IF (VI_Severity <> L_Last_Severity) OR (VI_RootCause <> L_Last_RootCause) THEN
    CASE VI_RootCause OF
        E_System_Root_Cause.ROOT_FIRE:
            L_Event_Text := 'EVENT: FIRE DETECTED';
        E_System_Root_Cause.ROOT_GAS_LEAK:
            L_Event_Text := 'EVENT: GAS LEAK';
        E_System_Root_Cause.ROOT_CO_CRITICAL:
            L_Event_Text := 'EVENT: CO CRITICAL';
        E_System_Root_Cause.ROOT_CO_WARNING:
            L_Event_Text := 'EVENT: CO WARNING';
        E_System_Root_Cause.ROOT_WATER_LEAK:
            L_Event_Text := 'EVENT: WATER LEAK';
        E_System_Root_Cause.ROOT_SENSOR_FAULT:
            L_Event_Text := 'EVENT: SENSOR FAULT';
        E_System_Root_Cause.ROOT_IO_OFFLINE:
            L_Event_Text := 'EVENT: IO OFFLINE';
        E_System_Root_Cause.ROOT_COMM_FAULT:
            L_Event_Text := 'EVENT: COMM FAULT';
        E_System_Root_Cause.ROOT_WATCHDOG_FAULT:
            L_Event_Text := 'EVENT: WATCHDOG FAULT';
        E_System_Root_Cause.ROOT_SUBSYSTEM_FAULT:
            L_Event_Text := 'EVENT: SUBSYSTEM FAULT';
        ELSE
            L_Event_Text := 'EVENT: SYSTEM STATE CHANGE';
    END_CASE;

    L_Write_Index := L_Write_Index + 1;
    IF L_Write_Index > 16 THEN
        L_Write_Index := 1;
    END_IF;

    VO_Event_Time_MS[L_Write_Index] := VI_Time_MS;
    VO_Event_Severity[L_Write_Index] := VI_Severity;
    VO_Event_RootCause[L_Write_Index] := VI_RootCause;
    VO_Event_Text[L_Write_Index] := L_Event_Text;

    VO_Last_Index := L_Write_Index;
    VO_Last_Event_Text := L_Event_Text;

    IF VO_Event_Count < 16 THEN
        VO_Event_Count := VO_Event_Count + 1;
    END_IF;
END_IF;

L_Last_Severity := VI_Severity;
L_Last_RootCause := VI_RootCause;
// >>> BULK_SYNC_ANCHOR: FB_Fault_Logger <<<

          
END_FUNCTION_BLOCK

FUNCTION_BLOCK FB_HMI_Interface
  VAR_INPUT
    VI_System_Time_MS : UDINT;
    VI_Latitude : REAL := 55.75;  (* Москва *)
    VI_Longitude : REAL := 37.61;
  END_VAR
  VAR_OUTPUT
    VO_Sunset_Time : TOD;
    VO_Sunrise_Time : TOD;
    VO_Is_Night : BOOL;
  END_VAR
  VAR
    L_Current_TOD : TOD;
  END_VAR

            FUNCTION_BLOCK FB_HMI_Interface
VAR_INPUT
    VI_Severity   : E_System_Severity;
    VI_RootCause  : E_System_Root_Cause;
    VI_Status_Msg : STRING(200);
END_VAR

VAR_OUTPUT
    VO_HMI_Status_Text : STRING(200);
    VO_HMI_State_Code  : INT;
END_VAR

VO_HMI_Status_Text := VI_Status_Msg;

CASE VI_Severity OF
    E_System_Severity.SEV_NORMAL:
        VO_HMI_State_Code := 0;
    E_System_Severity.SEV_WARNING:
        VO_HMI_State_Code := 1;
    E_System_Severity.SEV_DEGRADED:
        VO_HMI_State_Code := 2;
    E_System_Severity.SEV_CRITICAL:
        VO_HMI_State_Code := 3;
END_CASE;
// >>> BULK_SYNC_ANCHOR: FB_HMI_Interface <<<

          
END_FUNCTION_BLOCK

FUNCTION_BLOCK FB_IO_Module_Watchdog
  VAR_INPUT
    VI_System_Time_MS : UDINT;
    VI_Latitude : REAL := 55.75;  (* Москва *)
    VI_Longitude : REAL := 37.61;
  END_VAR
  VAR_OUTPUT
    VO_Sunset_Time : TOD;
    VO_Sunrise_Time : TOD;
    VO_Is_Night : BOOL;
  END_VAR
  VAR
    L_Current_TOD : TOD;
  END_VAR

            FUNCTION_BLOCK FB_IO_Module_Watchdog
VAR_INPUT
    VI_System_Time_MS : UDINT;
    VI_Module_ID : BYTE;
    VI_Heartbeat_Signal : BOOL; // Сигнал от модуля (например, мигающий бит)
    VI_Timeout_MS : UDINT := 2000; // Таймаут 2 секунды по умолчанию
END_VAR
VAR_OUTPUT
    VO_Module_Online : BOOL;
    VO_Error_Active : BOOL;
END_VAR
VAR
    L_Last_Heartbeat_State : BOOL;
    L_Last_Heartbeat_Time : UDINT;
    L_Elapsed_Time : UDINT;
END_VAR

// Отслеживание изменения сигнала
IF VI_Heartbeat_Signal <> L_Last_Heartbeat_State THEN
    L_Last_Heartbeat_Time := VI_System_Time_MS;
    L_Last_Heartbeat_State := VI_Heartbeat_Signal;
END_IF;

// Проверка таймаута
L_Elapsed_Time := F_TimeDiff(VI_System_Time_MS, L_Last_Heartbeat_Time);

IF L_Elapsed_Time > VI_Timeout_MS THEN
    VO_Module_Online := FALSE;
    VO_Error_Active := TRUE;
ELSE
    VO_Module_Online := TRUE;
    VO_Error_Active := FALSE;
END_IF;
// >>> BULK_SYNC_ANCHOR: FB_IO_Module_Watchdog <<<

          
END_FUNCTION_BLOCK

FUNCTION_BLOCK FB_Redundancy_Manager
  VAR_INPUT
    VI_System_Time_MS : UDINT;
    VI_Latitude : REAL := 55.75;  (* Москва *)
    VI_Longitude : REAL := 37.61;
  END_VAR
  VAR_OUTPUT
    VO_Sunset_Time : TOD;
    VO_Sunrise_Time : TOD;
    VO_Is_Night : BOOL;
  END_VAR
  VAR
    L_Current_TOD : TOD;
  END_VAR

            FUNCTION_BLOCK FB_Redundancy_Manager
VAR_INPUT
    VI_System_Time_MS : UDINT; // Системное время (мс)
    VI_Local_PLC_ID : BYTE; // 1 = ПЛК А, 2 = ПЛК B
    VI_Remote_Pulse : BOOL; // Сигнал от партнера
    VI_Remote_Is_Active : BOOL; // Статус партнера
    VI_Gateway_Ping_OK : BOOL; // Пинг до шлюза
    VI_Remote_State : ST_System_State_Snapshot; // Состояние партнера
    VI_Local_State : ST_System_State_Snapshot; // Локальное состояние
END_VAR
VAR_OUTPUT
    VO_Local_Role : E_PLC_ROLE; // Локальная роль ПЛК (Active/Standby)
    VO_Local_Pulse : BOOL; // Локальный сигнал пульса для партнера
    VO_Sync_Data_Req : BOOL; // Запрос на синхронизацию данных
    VO_Status_Msg : STRING(200); // Строковое сообщение о статусе
    VO_Synced_State : ST_System_State_Snapshot; // Синхронизированное состояние
    VO_State_Updated : BOOL; // Флаг: Состояние было обновлено
END_VAR
VAR
    L_Heartbeat : FB_PLC_Heartbeat;
    L_Pulse_Timer : FB_System_Timer;
    L_Pulse_State : BOOL;
    L_Prev_Role : E_PLC_ROLE;
    L_State_Replicator : FB_State_Replication;
END_VAR

// 1. Генерация собственного пульса (меандр 100 мс)
L_Pulse_Timer(IN := NOT L_Pulse_Timer.Q, PT := T#100ms, VI_System_Time_MS := VI_System_Time_MS);
IF L_Pulse_Timer.Q THEN
    L_Pulse_State := NOT L_Pulse_State;
END_IF;
VO_Local_Pulse := L_Pulse_State;

// 2. Определение роли через Heartbeat
L_Heartbeat(
    VI_Local_ID := VI_Local_PLC_ID,
    VI_System_Time := VI_System_Time_MS,
    VI_Remote_Pulse := VI_Remote_Pulse,
    VI_Remote_Is_Active := VI_Remote_Is_Active,
    VI_Gateway_Ping_OK := VI_Gateway_Ping_OK
);

IF L_Heartbeat.VO_Is_Active THEN
    VO_Local_Role := E_PLC_ROLE.ROLE_ACTIVE;
    VO_Status_Msg := 'ПЛК АКТИВЕН (ВЕДУЩИЙ)';
ELSE
    VO_Local_Role := E_PLC_ROLE.ROLE_STANDBY;
    VO_Status_Msg := 'ПЛК В РЕЗЕРВЕ (ВЕДОМЫЙ)';
END_IF;

// 3. Запрос на синхронизацию при переходе в ACTIVE
IF VO_Local_Role = E_PLC_ROLE.ROLE_ACTIVE AND L_Prev_Role = E_PLC_ROLE.ROLE_STANDBY THEN
    VO_Sync_Data_Req := TRUE;
ELSE
    VO_Sync_Data_Req := FALSE;
END_IF;

L_State_Replicator(
    VI_Local_Role := VO_Local_Role,
    VI_Sync_Req := VO_Sync_Data_Req,
    VI_Local_State := VI_Local_State,
    VI_Remote_State := VI_Remote_State,
    VI_System_Time_MS := VI_System_Time_MS
);
VO_Synced_State := L_State_Replicator.VO_Synced_State;
VO_State_Updated := L_State_Replicator.VO_State_Updated;

L_Prev_Role := VO_Local_Role;
// >>> BULK_SYNC_ANCHOR: FB_Redundancy_Manager <<<

          
END_FUNCTION_BLOCK

FUNCTION_BLOCK FB_Rule_Engine
  VAR_INPUT
    VI_System_Time_MS : UDINT;
    VI_Latitude : REAL := 55.75;  (* Москва *)
    VI_Longitude : REAL := 37.61;
  END_VAR
  VAR_OUTPUT
    VO_Sunset_Time : TOD;
    VO_Sunrise_Time : TOD;
    VO_Is_Night : BOOL;
  END_VAR
  VAR
    L_Current_TOD : TOD;
  END_VAR

            FUNCTION_BLOCK FB_Rule_Engine
VAR_INPUT
    VI_System_Time_MS : UDINT; // Системное время (мс)
    VI_IsActivePLC : BOOL; // Флаг: Данный ПЛК является ведущим
    VI_Security_Armed : BOOL; // Статус: Система под охраной
    VI_Current_Time : TOD; // Текущее время суток
    VI_Day_Of_Week : INT; // Текущий день недели (1..7, 1 = Понедельник)
END_VAR
VAR_IN_OUT
    VI_Rules : ARRAY[1..GVL_CONSTANTS.C_MAX_RULES] OF ST_User_Rule; // Массив пользовательских правил
    VI_Indoor_Temps : ARRAY[1..GVL_CONSTANTS.C_MAX_CLIMATE_ZONES] OF REAL; // Температуры в помещениях
    VI_Floor_Temps : ARRAY[1..GVL_CONSTANTS.C_MAX_HEATING_CIRCUITS] OF REAL; // Температуры пола
    VI_Humidities : ARRAY[1..GVL_CONSTANTS.C_MAX_CLIMATE_ZONES] OF REAL; // Влажность в помещениях
    VI_CO2_Levels : ARRAY[1..GVL_CONSTANTS.C_MAX_CLIMATE_ZONES] OF REAL; // Уровни CO2
    VI_Motion_Sensors : ARRAY[1..GVL_CONSTANTS.C_MAX_CLIMATE_ZONES] OF BOOL; // Датчики движения
    VI_Door_Sensors : ARRAY[1..GVL_CONSTANTS.C_MAX_DOOR_SENSORS] OF BOOL; // Датчики открытия дверей
    VI_Window_Sensors : ARRAY[1..GVL_CONSTANTS.C_MAX_CLIMATE_ZONES] OF BOOL; // Датчики открытия окон
    VI_Water_Sensors : ARRAY[1..GVL_CONSTANTS.C_MAX_FLOOD_SENSORS] OF BOOL; // Датчики протечки воды
    VI_Smoke_Sensors : ARRAY[1..GVL_CONSTANTS.C_MAX_SMOKE_SENSORS] OF BOOL; // Датчики дыма
    VI_Methane_Sensors : ARRAY[1..GVL_CONSTANTS.C_MAX_METHANE_SENSORS] OF REAL; // Датчики метана
    VI_CO_Sensors : ARRAY[1..GVL_CONSTANTS.C_MAX_CO_SENSORS] OF REAL; // Датчики угарного газа
END_VAR
VAR_OUTPUT
    VO_Actions : ARRAY[1..GVL_CONSTANTS.C_MAX_RULES] OF ST_Rule_Action; // Сформированные действия по правилам
END_VAR
VAR
    L_i : INT;
    fbCompat : ARRAY[1..GVL_CONSTANTS.C_MAX_RULES] OF FB_Rule_Compatibility_Package_DRAFT;
    L_Compat_All_OK : BOOL;
    L_Compat_First_Warning : STRING(255);
    L_Compat_First_Warning_Latched : BOOL;
    L_Shadow_V2_Enabled : BOOL;
    L_Shadow_V2_Roundtrip_Mismatch : BOOL;
    L_Shadow_V2_First_Mismatch_Rule : INT;
    L_V2_Switch_Enabled : BOOL;
    L_V2_Path_Ready : BOOL;
    L_V2_Using_Legacy_Fallback : BOOL;
    L_Condition_Met : BOOL;
    L_Current_Value : REAL;
    L_Triggers : ARRAY[1..GVL_CONSTANTS.C_MAX_RULES] OF R_TRIG;
    L_Trigger_Count : ARRAY[1..GVL_CONSTANTS.C_MAX_RULES] OF UINT;
    L_Last_Reset_Time : UDINT;
    L_Elapsed_Time : UDINT;
END_VAR

IF NOT VI_IsActivePLC THEN RETURN; END_IF;

L_Compat_All_OK := TRUE;
L_Compat_First_Warning := '';
L_Compat_First_Warning_Latched := FALSE;
L_Shadow_V2_Enabled := TRUE;
L_Shadow_V2_Roundtrip_Mismatch := FALSE;
L_Shadow_V2_First_Mismatch_Rule := 0;
L_V2_Switch_Enabled := FALSE;
L_V2_Path_Ready := FALSE;
L_V2_Using_Legacy_Fallback := TRUE;

// Сброс счетчиков срабатываний каждую минуту (защита от циклических зависимостей/дребезга)
L_Elapsed_Time := F_TimeDiff(VI_System_Time_MS, L_Last_Reset_Time);

IF L_Elapsed_Time >= GVL_CONSTANTS.C_MS_IN_MINUTE THEN
    L_Last_Reset_Time := VI_System_Time_MS;
    FOR L_i := 1 TO GVL_CONSTANTS.C_MAX_RULES DO
        L_Trigger_Count[L_i] := 0;
    END_FOR;
END_IF;

FOR L_i := 1 TO GVL_CONSTANTS.C_MAX_RULES DO
    fbCompat[L_i](VI_Rule_Legacy := VI_Rules[L_i]);

    IF NOT fbCompat[L_i].VO_Forward_OK OR NOT fbCompat[L_i].VO_Reverse_OK THEN
        L_Compat_All_OK := FALSE;
    END_IF;

    IF (NOT L_Compat_First_Warning_Latched) AND (fbCompat[L_i].VO_Warning_Text <> '') THEN
        L_Compat_First_Warning := fbCompat[L_i].VO_Warning_Text;
        L_Compat_First_Warning_Latched := TRUE;
    END_IF;

    IF L_Shadow_V2_Enabled THEN
        IF (fbCompat[L_i].VO_Rule_Legacy_Roundtrip.Action_Type <> VI_Rules[L_i].Action_Type)
           OR (fbCompat[L_i].VO_Rule_Legacy_Roundtrip.Action_Target_ID <> VI_Rules[L_i].Action_Target_ID)
           OR (ABS(fbCompat[L_i].VO_Rule_Legacy_Roundtrip.Action_Value - VI_Rules[L_i].Action_Value) > 0.0001)
           OR (fbCompat[L_i].VO_Rule_Legacy_Roundtrip.Condition_Type <> VI_Rules[L_i].Condition_Type)
           OR (fbCompat[L_i].VO_Rule_Legacy_Roundtrip.Condition_Target_ID <> VI_Rules[L_i].Condition_Target_ID)
           OR (fbCompat[L_i].VO_Rule_Legacy_Roundtrip.Condition_Op <> VI_Rules[L_i].Condition_Op)
           OR (ABS(fbCompat[L_i].VO_Rule_Legacy_Roundtrip.Condition_Value - VI_Rules[L_i].Condition_Value) > 0.0001)
           OR (ABS(fbCompat[L_i].VO_Rule_Legacy_Roundtrip.Condition_Value_Max - VI_Rules[L_i].Condition_Value_Max) > 0.0001) THEN
            L_Shadow_V2_Roundtrip_Mismatch := TRUE;
            IF L_Shadow_V2_First_Mismatch_Rule = 0 THEN
                L_Shadow_V2_First_Mismatch_Rule := L_i;
            END_IF;
        END_IF;
    END_IF;

    // Phase 4 scaffold: optional V2 switch point.
    // Current state: always remain on legacy behavior.
    // Future state: when V2 path is implemented and validated,
    // this block becomes the controlled branch point.
    IF L_V2_Switch_Enabled AND L_V2_Path_Ready THEN
        L_V2_Using_Legacy_Fallback := FALSE;
        // V2 action-generation path placeholder.
        // No runtime behavior change yet.
    ELSE
        L_V2_Using_Legacy_Fallback := TRUE;
    END_IF;

    VO_Actions[L_i].Active := FALSE;
    IF VI_Rules[L_i].Enabled THEN
        L_Condition_Met := FALSE;
        L_Current_Value := 0.0;
        
        // Определение значения для проверки
        IF VI_Rules[L_i].Condition_Target_ID > 0 THEN
            CASE VI_Rules[L_i].Condition_Type OF
                E_Rule_Condition_Type.COND_AIR_TEMP: IF VI_Rules[L_i].Condition_Target_ID <= GVL_CONSTANTS.C_MAX_CLIMATE_ZONES THEN L_Current_Value := VI_Indoor_Temps[VI_Rules[L_i].Condition_Target_ID]; END_IF;
                E_Rule_Condition_Type.COND_FLOOR_TEMP: IF VI_Rules[L_i].Condition_Target_ID <= GVL_CONSTANTS.C_MAX_HEATING_CIRCUITS THEN L_Current_Value := VI_Floor_Temps[VI_Rules[L_i].Condition_Target_ID]; END_IF;
                E_Rule_Condition_Type.COND_HUMIDITY: IF VI_Rules[L_i].Condition_Target_ID <= GVL_CONSTANTS.C_MAX_CLIMATE_ZONES THEN L_Current_Value := VI_Humidities[VI_Rules[L_i].Condition_Target_ID]; END_IF;
                E_Rule_Condition_Type.COND_CO2: IF VI_Rules[L_i].Condition_Target_ID <= GVL_CONSTANTS.C_MAX_CLIMATE_ZONES THEN L_Current_Value := VI_CO2_Levels[VI_Rules[L_i].Condition_Target_ID]; END_IF;
                E_Rule_Condition_Type.COND_MOTION: IF VI_Rules[L_i].Condition_Target_ID <= GVL_CONSTANTS.C_MAX_CLIMATE_ZONES THEN L_Current_Value := SEL(VI_Motion_Sensors[VI_Rules[L_i].Condition_Target_ID], 0.0, 1.0); END_IF;
                E_Rule_Condition_Type.COND_DOOR_WINDOW: 
                    IF VI_Rules[L_i].Condition_Target_ID <= GVL_CONSTANTS.C_MAX_DOOR_SENSORS THEN
                        L_Current_Value := SEL(VI_Door_Sensors[VI_Rules[L_i].Condition_Target_ID] OR VI_Window_Sensors[VI_Rules[L_i].Condition_Target_ID], 0.0, 1.0);
                    ELSIF VI_Rules[L_i].Condition_Target_ID <= GVL_CONSTANTS.C_MAX_CLIMATE_ZONES THEN
                        L_Current_Value := SEL(VI_Window_Sensors[VI_Rules[L_i].Condition_Target_ID], 0.0, 1.0);
                    END_IF;
                E_Rule_Condition_Type.COND_FLOOD: IF VI_Rules[L_i].Condition_Target_ID <= GVL_CONSTANTS.C_MAX_FLOOD_SENSORS THEN L_Current_Value := SEL(VI_Water_Sensors[VI_Rules[L_i].Condition_Target_ID], 0.0, 1.0); END_IF;
                E_Rule_Condition_Type.COND_SMOKE: IF VI_Rules[L_i].Condition_Target_ID <= GVL_CONSTANTS.C_MAX_SMOKE_SENSORS THEN L_Current_Value := SEL(VI_Smoke_Sensors[VI_Rules[L_i].Condition_Target_ID], 0.0, 1.0); END_IF;
                E_Rule_Condition_Type.COND_METHANE: IF VI_Rules[L_i].Condition_Target_ID <= GVL_CONSTANTS.C_MAX_METHANE_SENSORS THEN L_Current_Value := VI_Methane_Sensors[VI_Rules[L_i].Condition_Target_ID]; END_IF;
                E_Rule_Condition_Type.COND_CO: IF VI_Rules[L_i].Condition_Target_ID <= GVL_CONSTANTS.C_MAX_CO_SENSORS THEN L_Current_Value := VI_CO_Sensors[VI_Rules[L_i].Condition_Target_ID]; END_IF;
                E_Rule_Condition_Type.COND_TIME_OF_DAY: L_Current_Value := TO_REAL(TOD_TO_UDINT(VI_Current_Time) / GVL_CONSTANTS.C_MS_IN_MINUTE); // Время в минутах
                E_Rule_Condition_Type.COND_DAY_OF_WEEK: L_Current_Value := TO_REAL(VI_Day_Of_Week);
            END_CASE;
        ELSE
            IF VI_Rules[L_i].Condition_Type = E_Rule_Condition_Type.COND_TIME_OF_DAY THEN
                L_Current_Value := TO_REAL(TOD_TO_UDINT(VI_Current_Time) / GVL_CONSTANTS.C_MS_IN_MINUTE); // Время в минутах
            ELSIF VI_Rules[L_i].Condition_Type = E_Rule_Condition_Type.COND_DAY_OF_WEEK THEN
                L_Current_Value := TO_REAL(VI_Day_Of_Week);
            END_IF;
        END_IF;
        
        // Проверка условия
        CASE VI_Rules[L_i].Condition_Op OF
            E_Rule_Comparison.COMP_GT: L_Condition_Met := (L_Current_Value > VI_Rules[L_i].Condition_Value);
            E_Rule_Comparison.COMP_LT: L_Condition_Met := (L_Current_Value < VI_Rules[L_i].Condition_Value);
            E_Rule_Comparison.COMP_EQ: L_Condition_Met := (ABS(L_Current_Value - VI_Rules[L_i].Condition_Value) < 0.1);
            E_Rule_Comparison.COMP_GE: L_Condition_Met := (L_Current_Value >= VI_Rules[L_i].Condition_Value);
            E_Rule_Comparison.COMP_LE: L_Condition_Met := (L_Current_Value <= VI_Rules[L_i].Condition_Value);
            E_Rule_Comparison.COMP_IN_RANGE: L_Condition_Met := (L_Current_Value >= VI_Rules[L_i].Condition_Value) AND (L_Current_Value <= VI_Rules[L_i].Condition_Value_Max);
            E_Rule_Comparison.COMP_TRUE: L_Condition_Met := (L_Current_Value > 0.5);
            E_Rule_Comparison.COMP_FALSE: L_Condition_Met := (L_Current_Value < 0.5);
        END_CASE;
        
        // Формирование действия
        L_Triggers[L_i](CLK := L_Condition_Met);
        
        IF L_Triggers[L_i].Q THEN
            L_Trigger_Count[L_i] := L_Trigger_Count[L_i] + 1;
            IF L_Trigger_Count[L_i] > 10 THEN
                // ТЗ 13.5: Блокировка правила при слишком частом срабатывании (циклическая зависимость)
                VO_Actions[L_i].Active := FALSE;
                VO_Actions[L_i].Triggered := FALSE;
                CONTINUE; // Пропускаем выполнение
            END_IF;
        END_IF;
        
        IF L_Condition_Met AND (L_Trigger_Count[L_i] <= 10) THEN
            VO_Actions[L_i].Active := TRUE;
            VO_Actions[L_i].Triggered := L_Triggers[L_i].Q;
            VO_Actions[L_i].Action_Type := VI_Rules[L_i].Action_Type;
            VO_Actions[L_i].Target_ID := VI_Rules[L_i].Action_Target_ID;
            VO_Actions[L_i].Value := VI_Rules[L_i].Action_Value;
        END_IF;
    END_IF;
END_FOR;
// >>> BULK_SYNC_ANCHOR: FB_Rule_Engine <<<

          
END_FUNCTION_BLOCK

FUNCTION_BLOCK FB_Safety_Manager
  VAR_INPUT
    VI_System_Time_MS : UDINT;
    VI_Latitude : REAL := 55.75;  (* Москва *)
    VI_Longitude : REAL := 37.61;
  END_VAR
  VAR_OUTPUT
    VO_Sunset_Time : TOD;
    VO_Sunrise_Time : TOD;
    VO_Is_Night : BOOL;
  END_VAR
  VAR
    L_Current_TOD : TOD;
  END_VAR

            FUNCTION_BLOCK FB_Safety_Manager
VAR_INPUT
    VI_Gas_Alarm : BOOL;
    VI_Leak_Alarm : BOOL;
    VI_Smoke_Alarm : BOOL;
    VI_Reset : BOOL; // Ручной сброс защёлкнутых safety-аварий оператором
END_VAR
VAR_OUTPUT
    VO_Gas_Latched : BOOL;
    VO_Leak_Latched : BOOL;
    VO_Smoke_Latched : BOOL;
    VO_Emergency_Stop : BOOL;
END_VAR
VAR
    L_Any_Active : BOOL;
END_VAR

// Защёлкиваем аварии независимо друг от друга
IF VI_Gas_Alarm THEN
    VO_Gas_Latched := TRUE;
END_IF;

IF VI_Leak_Alarm THEN
    VO_Leak_Latched := TRUE;
END_IF;

IF VI_Smoke_Alarm THEN
    VO_Smoke_Latched := TRUE;
END_IF;

L_Any_Active := VI_Gas_Alarm OR VI_Leak_Alarm OR VI_Smoke_Alarm;

// Ручной сброс допустим только когда все входные аварийные сигналы уже исчезли
IF VI_Reset AND NOT L_Any_Active THEN
    VO_Gas_Latched := FALSE;
    VO_Leak_Latched := FALSE;
    VO_Smoke_Latched := FALSE;
END_IF;

// Агрегированный аварийный стоп = любая защёлкнутая safety-авария
VO_Emergency_Stop := VO_Gas_Latched OR VO_Leak_Latched OR VO_Smoke_Latched;
END_FUNCTION_BLOCK
// >>> BULK_SYNC_ANCHOR: FB_Safety_Manager <<<

          
END_FUNCTION_BLOCK

FUNCTION_BLOCK FB_Socket_Manager
  VAR_INPUT
    VI_System_Time_MS : UDINT;
    VI_Latitude : REAL := 55.75;  (* Москва *)
    VI_Longitude : REAL := 37.61;
  END_VAR
  VAR_OUTPUT
    VO_Sunset_Time : TOD;
    VO_Sunrise_Time : TOD;
    VO_Is_Night : BOOL;
  END_VAR
  VAR
    L_Current_TOD : TOD;
  END_VAR

            FUNCTION_BLOCK FB_Socket_Manager
// Менеджер управления розетками.
// Обеспечивает работу по сценариям, правилам и аварийное отключение (без локальных выключателей розеток).
VAR_INPUT
    VI_System_Time_MS : UDINT; // Системное время в миллисекундах
    VI_IsActivePLC : BOOL; // Флаг активности ПЛК (TRUE = ведущий)
    VI_Scenario : E_SCENARIO_TYPE; // Текущий глобальный сценарий
    VI_Fire_Alarm : BOOL; // Флаг пожарной тревоги
    VI_Flood_Alarm : BOOL; // Флаг тревоги протечки
    VI_Security_Armed : BOOL; // Состояние охраны (TRUE = включена)
END_VAR
VAR_IN_OUT
    VI_Manual_Override : ARRAY[1..GVL_CONSTANTS.C_MAX_SOCKETS] OF BOOL; // Ручное переопределение состояния (HMI)
    VI_Physical_Switches : ARRAY[1..GVL_CONSTANTS.C_MAX_SOCKETS] OF BOOL; // Legacy-вход: не используется в текущей концепции
    VI_Rule_Actions : ARRAY[1..GVL_CONSTANTS.C_MAX_RULES] OF ST_Rule_Action; // Действия от Rule Engine
    VI_IO_Modules_Online : ARRAY[1..GVL_CONSTANTS.C_MAX_MODULES] OF BOOL; // Статусы модулей ввода-вывода
END_VAR
VAR_OUTPUT
    VO_Socket_States : ARRAY[1..GVL_CONSTANTS.C_MAX_SOCKETS] OF BOOL; // Выходные состояния розеток
    VO_Internal_States : ARRAY[1..GVL_CONSTANTS.C_MAX_SOCKETS] OF BOOL; // Внутренние состояния для репликации
END_VAR
VAR
    // Socket V2 shadow (phase2)
    fbSocketV2Staging : FB_Socket_V2_Staging_DRAFT;
    L_Socket_V2_Command_Shadow : ST_Socket_Command_V2;
    L_Socket_V2_State_Shadow : ST_Socket_State_V2;
    L_Socket_V2_Shadow_Diff_Found : BOOL;
    L_Socket_V2_Switch_Enabled : BOOL;
    L_Socket_V2_Path_Ready : BOOL;
    L_Socket_Using_Legacy_Fallback : BOOL;
    L_i : INT;
    L_j : INT;
    L_Rule_State : BOOL;
    L_Rule_Active : BOOL;
    L_Internal_State : ARRAY[1..GVL_CONSTANTS.C_MAX_SOCKETS] OF BOOL;
    L_Manual_Trig : ARRAY[1..GVL_CONSTANTS.C_MAX_SOCKETS] OF R_TRIG;
END_VAR

IF NOT VI_IsActivePLC THEN RETURN; END_IF;

L_Socket_V2_Shadow_Diff_Found := FALSE;
L_Socket_V2_Switch_Enabled := TRUE;
L_Socket_V2_Path_Ready := FALSE;
L_Socket_Using_Legacy_Fallback := TRUE;

// Проверка связи с модулями ввода-вывода
FOR L_i := 1 TO GVL_CONSTANTS.C_MAX_MODULES DO
    IF NOT VI_IO_Modules_Online[L_i] THEN
        // Переход в безопасное состояние при потере связи (отключение всех розеток)
        FOR L_j := 1 TO GVL_CONSTANTS.C_MAX_SOCKETS DO
            VO_Socket_States[L_j] := FALSE;
        END_FOR;
        RETURN;
    END_IF;
END_FOR;

FOR L_i := 1 TO GVL_CONSTANTS.C_MAX_SOCKETS DO
    L_Rule_Active := FALSE;
    L_Rule_State := FALSE;
    
    L_Manual_Trig[L_i](CLK := VI_Manual_Override[L_i]);
    
    // Ручное переключение
    IF L_Manual_Trig[L_i].Q THEN
        L_Internal_State[L_i] := NOT L_Internal_State[L_i];
    END_IF;

    // Проверка правил для текущей розетки
    FOR L_j := 1 TO GVL_CONSTANTS.C_MAX_RULES DO
        IF VI_Rule_Actions[L_j].Active AND VI_Rule_Actions[L_j].Target_ID = L_i THEN
            IF VI_Rule_Actions[L_j].Action_Type = E_Rule_Action_Type.ACTION_SET_SOCKET THEN
                L_Rule_Active := TRUE;
                L_Rule_State := (VI_Rule_Actions[L_j].Value > 0.5);
                L_Internal_State[L_i] := L_Rule_State; // Синхронизация внутреннего состояния
            ELSIF VI_Rule_Actions[L_j].Action_Type = E_Rule_Action_Type.ACTION_TOGGLE_SOCKET AND VI_Rule_Actions[L_j].Triggered THEN
                L_Internal_State[L_i] := NOT L_Internal_State[L_i]; // Toggle
            END_IF;
        END_IF;
    END_FOR;

    // Аварийное отключение
    IF VI_Fire_Alarm OR VI_Flood_Alarm THEN
        // Розетки 1-4 неотключаемые (холодильник, сервер и т.д.)
        IF L_i > 4 THEN
            VO_Socket_States[L_i] := FALSE;
        ELSE
            // Критические розетки сохраняют свое текущее внутреннее состояние, а не форсируются в TRUE
            VO_Socket_States[L_i] := L_Internal_State[L_i];
        END_IF;
    ELSIF VI_Scenario = E_SCENARIO_TYPE.SCENARIO_AWAY OR VI_Security_Armed THEN
        // Master Off
        IF L_i > 4 THEN
            VO_Socket_States[L_i] := FALSE;
        ELSE
            // Неотключаемые розетки могут управляться вручную
            VO_Socket_States[L_i] := L_Internal_State[L_i];
        END_IF;
    ELSE
        // Нормальный режим: состояние определяется внутренним состоянием (ручным или правилом)
        IF L_Rule_Active THEN
            VO_Socket_States[L_i] := L_Rule_State;
        ELSE
            VO_Socket_States[L_i] := L_Internal_State[L_i];
        END_IF;
    END_IF;
END_FOR;

VO_Internal_States := L_Internal_State;

// ========================================
// Socket V2 shadow execution (phase2)
// ========================================
fbSocketV2Staging(
    VI_Socket_ID := 1,
    VI_Enable := TRUE,
    VI_Target_State := VO_Socket_States[1],
    VI_Manual_Override := VI_Manual_Override[1],
    VI_Safety_Lock := (VI_Fire_Alarm OR VI_Flood_Alarm),
    VI_Scenario_ID := TO_INT(VI_Scenario),

    VI_Is_On := VO_Socket_States[1],
    VI_Manual_Override_Active := VI_Manual_Override[1],
    VI_Safety_Blocked := (VI_Fire_Alarm OR VI_Flood_Alarm),
    VI_Alarm_Active := (VI_Fire_Alarm OR VI_Flood_Alarm),

    VO_Command_Shadow => L_Socket_V2_Command_Shadow,
    VO_State_Shadow => L_Socket_V2_State_Shadow
);

// ========================================
// Socket V2 shadow validation
// ========================================
IF VO_Socket_States[1] <> L_Socket_V2_Command_Shadow.Target_State THEN
    L_Socket_V2_Shadow_Diff_Found := TRUE;
END_IF;
IF VO_Socket_States[1] <> L_Socket_V2_State_Shadow.Is_On THEN
    L_Socket_V2_Shadow_Diff_Found := TRUE;
END_IF;
IF (VI_Fire_Alarm OR VI_Flood_Alarm) <> L_Socket_V2_State_Shadow.Safety_Blocked THEN
    L_Socket_V2_Shadow_Diff_Found := TRUE;
END_IF;

// Guarded Socket V2 enable
IF L_Socket_V2_Switch_Enabled THEN
    IF NOT L_Socket_V2_Shadow_Diff_Found THEN
        L_Socket_V2_Path_Ready := TRUE;
        L_Socket_Using_Legacy_Fallback := FALSE;
    ELSE
        L_Socket_V2_Path_Ready := FALSE;
        L_Socket_Using_Legacy_Fallback := TRUE;
    END_IF;
ELSE
    L_Socket_V2_Path_Ready := FALSE;
    L_Socket_Using_Legacy_Fallback := TRUE;
END_IF;

END_FUNCTION_BLOCK
// >>> BULK_SYNC_ANCHOR: FB_Socket_Manager <<<

          
END_FUNCTION_BLOCK

FUNCTION_BLOCK FB_System_Health
  VAR_INPUT
    VI_System_Time_MS : UDINT;
    VI_Latitude : REAL := 55.75;  (* Москва *)
    VI_Longitude : REAL := 37.61;
  END_VAR
  VAR_OUTPUT
    VO_Sunset_Time : TOD;
    VO_Sunrise_Time : TOD;
    VO_Is_Night : BOOL;
  END_VAR
  VAR
    L_Current_TOD : TOD;
  END_VAR

            FUNCTION_BLOCK FB_System_Health
VAR_INPUT
    VI_Smoke_Detected      : BOOL;
    VI_Gas_Detected        : BOOL;
    VI_CO_Warning_Level    : BOOL;
    VI_CO_Alarm_Level      : BOOL;
    VI_Leak_Detected       : BOOL;

    VI_Sensor_Fault        : BOOL := FALSE;
    VI_IO_Offline          : BOOL := FALSE;
    VI_Comm_Fault          : BOOL := FALSE;
    VI_Watchdog_Fault      : BOOL := FALSE;
    VI_Subsystem_Fault     : BOOL := FALSE;
END_VAR

VAR_OUTPUT
    VO_System_Severity     : E_System_Severity;
    VO_Root_Cause          : E_System_Root_Cause;

    // compatibility outputs for existing orchestration
    VO_Sensor_Fault        : BOOL;
    VO_IO_Fault            : BOOL;
    VO_Comm_Fault          : BOOL;
    VO_Subsystem_Degraded  : BOOL;

    VO_First_Fault_Active  : BOOL;
    VO_First_Fault_Type    : INT;
    VO_First_Fault_Source  : INT;
END_VAR

VO_Sensor_Fault := VI_Sensor_Fault;
VO_IO_Fault := VI_IO_Offline;
VO_Comm_Fault := VI_Comm_Fault;
VO_Subsystem_Degraded := VI_Subsystem_Fault;

VO_System_Severity := E_System_Severity.SEV_NORMAL;
VO_Root_Cause := E_System_Root_Cause.ROOT_NONE;
VO_First_Fault_Active := FALSE;
VO_First_Fault_Type := 0;
VO_First_Fault_Source := 0;

// Priority: FIRE > GAS > CO > WATER > diagnostics
IF VI_Smoke_Detected THEN
    VO_System_Severity := E_System_Severity.SEV_CRITICAL;
    VO_Root_Cause := E_System_Root_Cause.ROOT_FIRE;
    VO_First_Fault_Active := TRUE;
    VO_First_Fault_Type := 5;

ELSIF VI_Gas_Detected THEN
    VO_System_Severity := E_System_Severity.SEV_CRITICAL;
    VO_Root_Cause := E_System_Root_Cause.ROOT_GAS_LEAK;
    VO_First_Fault_Active := TRUE;
    VO_First_Fault_Type := 6;

ELSIF VI_CO_Alarm_Level THEN
    VO_System_Severity := E_System_Severity.SEV_CRITICAL;
    VO_Root_Cause := E_System_Root_Cause.ROOT_CO_CRITICAL;
    VO_First_Fault_Active := TRUE;
    VO_First_Fault_Type := 7;

ELSIF VI_CO_Warning_Level THEN
    VO_System_Severity := E_System_Severity.SEV_WARNING;
    VO_Root_Cause := E_System_Root_Cause.ROOT_CO_WARNING;
    VO_First_Fault_Active := TRUE;
    VO_First_Fault_Type := 7;

ELSIF VI_Leak_Detected THEN
    VO_System_Severity := E_System_Severity.SEV_WARNING;
    VO_Root_Cause := E_System_Root_Cause.ROOT_WATER_LEAK;
    VO_First_Fault_Active := TRUE;
    VO_First_Fault_Type := 8;

ELSIF VI_Watchdog_Fault THEN
    VO_System_Severity := E_System_Severity.SEV_CRITICAL;
    VO_Root_Cause := E_System_Root_Cause.ROOT_WATCHDOG_FAULT;
    VO_First_Fault_Active := TRUE;
    VO_First_Fault_Type := 9;

ELSIF VI_IO_Offline THEN
    VO_System_Severity := E_System_Severity.SEV_DEGRADED;
    VO_Root_Cause := E_System_Root_Cause.ROOT_IO_OFFLINE;
    VO_First_Fault_Active := TRUE;
    VO_First_Fault_Type := 1;

ELSIF VI_Comm_Fault THEN
    VO_System_Severity := E_System_Severity.SEV_DEGRADED;
    VO_Root_Cause := E_System_Root_Cause.ROOT_COMM_FAULT;
    VO_First_Fault_Active := TRUE;
    VO_First_Fault_Type := 3;

ELSIF VI_Sensor_Fault THEN
    VO_System_Severity := E_System_Severity.SEV_DEGRADED;
    VO_Root_Cause := E_System_Root_Cause.ROOT_SENSOR_FAULT;
    VO_First_Fault_Active := TRUE;
    VO_First_Fault_Type := 2;

ELSIF VI_Subsystem_Fault THEN
    VO_System_Severity := E_System_Severity.SEV_DEGRADED;
    VO_Root_Cause := E_System_Root_Cause.ROOT_SUBSYSTEM_FAULT;
    VO_First_Fault_Active := TRUE;
    VO_First_Fault_Type := 4;
END_IF;
// >>> BULK_SYNC_ANCHOR: FB_System_Health <<<

          
END_FUNCTION_BLOCK

FUNCTION_BLOCK FB_System_Timer
  VAR_INPUT
    VI_System_Time_MS : UDINT;
    VI_Latitude : REAL := 55.75;  (* Москва *)
    VI_Longitude : REAL := 37.61;
  END_VAR
  VAR_OUTPUT
    VO_Sunset_Time : TOD;
    VO_Sunrise_Time : TOD;
    VO_Is_Night : BOOL;
  END_VAR
  VAR
    L_Current_TOD : TOD;
  END_VAR

            // ==============================================================================
// Блок таймера, привязанный к системному времени (System Timer)
// Назначение:
// - Замена стандартного TON для обеспечения точной выдержки времени,
//   независимой от времени цикла ПЛК, с использованием единого системного времени.
// ==============================================================================
FUNCTION_BLOCK FB_System_Timer
VAR_INPUT
    IN : BOOL; // Вход запуска таймера
    PT : TIME; // Заданное время
    VI_System_Time_MS : UDINT; // Системное время (мс)
END_VAR
VAR_OUTPUT
    Q : BOOL; // Выход: таймер сработал
    ET : TIME; // Прошедшее время
END_VAR
VAR
    L_Start_Time : UDINT;
    L_Running : BOOL;
END_VAR

IF IN THEN
    IF NOT L_Running THEN
        L_Start_Time := VI_System_Time_MS;
        L_Running := TRUE;
        ET := T#0s;
        Q := FALSE;
    ELSE
        // Обработка переполнения UDINT (примерно 49 дней)
        ET := TO_TIME(F_TimeDiff(VI_System_Time_MS, L_Start_Time));
        
        IF ET >= PT THEN
            Q := TRUE;
            ET := PT;
        ELSE
            Q := FALSE;
        END_IF;
    END_IF;
ELSE
    L_Running := FALSE;
    ET := T#0s;
    Q := FALSE;
END_IF;
// >>> BULK_SYNC_ANCHOR: FB_System_Timer <<<

          
END_FUNCTION_BLOCK

FUNCTION_BLOCK FB_Watchdog
  VAR_INPUT
    VI_System_Time_MS : UDINT;
    VI_Latitude : REAL := 55.75;  (* Москва *)
    VI_Longitude : REAL := 37.61;
  END_VAR
  VAR_OUTPUT
    VO_Sunset_Time : TOD;
    VO_Sunrise_Time : TOD;
    VO_Is_Night : BOOL;
  END_VAR
  VAR
    L_Current_TOD : TOD;
  END_VAR

            FUNCTION_BLOCK FB_Watchdog
VAR_INPUT
    VI_System_Time_MS : UDINT;
    VI_Timeout_MS     : UDINT := 2000;
END_VAR

VAR_OUTPUT
    VO_Alive          : BOOL;
    VO_Watchdog_Fault : BOOL;
    VO_Cycle_DT_MS    : UDINT;
END_VAR

VAR
    L_Initialized    : BOOL := FALSE;
    L_Last_Call_MS   : UDINT := 0;
    L_DT_MS          : UDINT := 0;
END_VAR

IF NOT L_Initialized THEN
    L_Initialized := TRUE;
    L_Last_Call_MS := VI_System_Time_MS;
    VO_Cycle_DT_MS := 0;
    VO_Watchdog_Fault := FALSE;
    VO_Alive := TRUE;
    RETURN;
END_IF;

// Measure real time gap between successive calls
L_DT_MS := F_TimeDiff(VI_System_Time_MS, L_Last_Call_MS);
VO_Cycle_DT_MS := L_DT_MS;

// Fault if the task/cycle resumed after an abnormal pause
VO_Watchdog_Fault := (L_DT_MS > VI_Timeout_MS);
VO_Alive := NOT VO_Watchdog_Fault;

// Store current timestamp for next cycle
L_Last_Call_MS := VI_System_Time_MS;
// >>> BULK_SYNC_ANCHOR: FB_Watchdog <<<

          
END_FUNCTION_BLOCK
